FUNCTION_BLOCK E_FB_TimeOut (* Simple implementation of the timeout services *)
  (* Standard: 61499-1; Description: Copyright (c) 2017 fortiss GmbH This program and the accompanying materials are made available under the terms of the Eclipse Public License 2.0 which is available at https://www.eclipse.org/legal/epl-2.0/ SPDX-License-Identifier: EPL-2.0 *)
  (* Version 3.1, 2026-08-14, Franz Höpfinger, HR Agrartechnik GmbH, FB_TON like cyclic Interface *)
  (* Version 3.0, 2025-04-14, Patrick Aigner, changed package *)
  (* Version 1.0, 2017-09-22, Alois Zoitl, fortiss GmbH, initial API and implementation and/or initial documentation *)
  PACKAGE adapter::events::TimeOut;
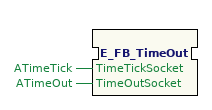
  SOCKETS
    TimeTickSocket : adapter::events::TimeOut::ATimeTick;
    TimeOutSocket : iec61499::events::ATimeOut;
  END_SOCKETS
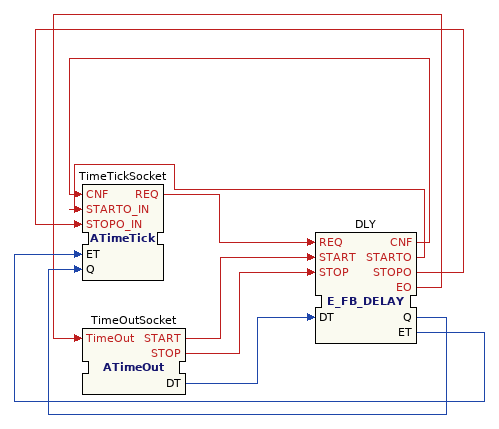
  FBS
    DLY : adapter::events::TimeOut::E_FB_DELAY;
  END_FBS
  EVENT_CONNECTIONS
    TimeOutSocket.START TO DLY.START;
    TimeOutSocket.STOP TO DLY.STOP;
    DLY.EO TO TimeOutSocket.TimeOut;
    TimeTickSocket.REQ TO DLY.REQ;
    DLY.CNF TO TimeTickSocket.CNF;
    DLY.STARTO TO TimeTickSocket.STARTO_IN;
    DLY.STOPO TO TimeTickSocket.STOPO_IN;
  END_CONNECTIONS
  DATA_CONNECTIONS
    TimeOutSocket.DT TO DLY.DT;
    DLY.ET TO TimeTickSocket.ET;
    DLY.Q TO TimeTickSocket.Q;
  END_CONNECTIONS
END_FUNCTION_BLOCK
